FUNCTION_BLOCK NodeFactory_Display_BOOL EXTENDS NodeFactory

METHOD PUBLIC Create : I_Node
VAR
	pointerToNode : POINTER TO Node_Display_BOOL;
END_VAR
pointerToNode := __NEW(Node_Display_BOOL);
Create := pointerToNode^;
END_METHOD

END_FUNCTION_BLOCK

(* stored: Version 1.1.0.1, ProductVersion 3.1.4024.12
   POU NodeFactory_Display_BOOL: Id {5cad8499-d6c8-0118-1afc-cd1bcbf5b9ae}, SpecialFunc None
   Method Create: Id {033e8683-3b32-0af1-3303-11473673c1cc} *)
